(* PLC project single_acting_rod, Dassault Systèmes ControlBuild 2024x *)
(* stored: creationDateTime 2023-10-03T11:13:16-01:00 *)

(* This modules simulates the bahaviour of a single-acting cylinder rod according to the state of pipes. *)
FUNCTION_BLOCK equipment_library.single_acting_rod
  VAR_INPUT
    pipeWork : BOOL := false;
  END_VAR
  VAR_OUTPUT
    rodPosition : REAL := 0.0;
    rodPercent : REAL := 0.0;
  END_VAR
  VAR
    increment : REAL := 0.0;
  END_VAR
  VAR CONSTANT
    length : REAL := 1000.0;
    timeOutput : REAL := 10.0;
  END_VAR
  VAR
    d_locking : BOOL := false;
    v_d_locking : REAL := 10.0;
  END_VAR


ACTION C_source_code:
/* ----------------------------------------------------------------	*/
/* Type : Model of Operative Behaviour					*/
/* Category :  Actuators							*/
/* Author : Dassault Systemes						*/
/* Update date : June 2018							*/
/* ----------------------------------------------------------------	*/
/* This module simulates the behaviour of a single-acting cylinder	*/
/* rod according to the working state of pipe.				*/
/* ----------------------------------------------------------------	*/

if (d_locking) increment=0;
else {
	increment=(length/timeOutput)*(CLOCK_PERIOD/1000000);
	if (pipeWork) {
		if ( rodPosition < length ) (rodPosition)+= increment;
		if ( rodPosition > length ) rodPosition = length;
	}
	else {
		if ( rodPosition > 0 ) (rodPosition)-= increment;
		if ( rodPosition < 0 ) rodPosition = 0;
	}
}

/* ----------------------------------------------------------------	*/
/* Compute the percentage of cylinder rod's length			*/
/* ----------------------------------------------------------------	*/
if (length > 0.0)
	rodPercent = ((rodPosition/length)*100);
END_ACTION
END_FUNCTION_BLOCK
